{attribute 'GeneratedUsingTerminal: EL1258-0000-0016'}
{attribute addProperty BoxType "EL1258-0000-0016"}
{attribute addProperty Id "CtrlAT %Q*Ctrl_F19EAB212"}
{attribute addProperty CRC "252717217"}
{attribute addProperty Size "2"}
TYPE MTI_Outputs_Channel_0F1028A1 EXTENDS OutputBase_10CEE7DE :
STRUCT
	{attribute addProperty Name "Ctrl"}
	Ctrl AT %Q* : Ctrl_F19EAB21;
END_STRUCT
END_TYPE

(* stored: Version 1.2.0.0, ProductVersion 3.1.4024.9
   DUT MTI_Outputs_Channel_0F1028A1: Id {96b36e22-74db-40bf-bacf-eb650f6d7236} *)
